
// ===== library: MasterCopy "TimerLibrary" =====

// folder: Timer Library

DATA_BLOCK "TimerLibraryVar"   // DB1
{ S7_Optimized_Access := 'TRUE' }
VERSION : 0.1
   VAR
      POS : Array[0..20] of Struct
         StopMode : Bool;
         ManualMode : Bool;
         AutoMode : Bool;
         CurrentEngineStatus : Int;
         TimeElapsed : Time;
         TimerTime : Time;
         TimerReset : Bool;
         TimerPreset : Bool;
      END_STRUCT;
      HmiPosition : Int := 1;
      ArrayPos : Int;
      Hmi : Struct
         ManualButton : Bool;
         StopButton : Bool;
         AutoButton : Bool;
         TiempoTrans : Time;
      END_STRUCT;
      Temp : Array[0..20] of Struct
         MotorTimer : TP_TIME;
      END_STRUCT;
   END_VAR
BEGIN
   Temp[1].MotorTimer.PT := T#1m;
   Temp[2].MotorTimer.PT := T#2m;
   Temp[3].MotorTimer.PT := T#3m;
   POS[2].TimerTime := T#2m;
   POS[1].TimerTime := T#1m;
   POS[3].TimerTime := T#3m;
END_DATA_BLOCK

FUNCTION "HmiButtonFunction" : Void   // FC4, SCL
{ S7_Optimized_Access := 'TRUE' }
VERSION : 0.1
BEGIN
   (*************************************************************************************************************
                                                 Function Block: Buttons and Operating Modes
   **************************************************************************************************************

   *    Project: Multiple Timer.
   *    Equipment: Siemens S7 1200 PLC
   *    Description: Function and programming of operating modes 
   *    Date: 18/01/2024

   **************************************************************************************************************)


   (* INSERT THIS CODE INTO THE MAIN BLOCK
           "TimerLibraryVar".ArrayPos := "TimerLibraryVar".ArrayPos + 1;
           IF "TimerLibraryVar".ArrayPos > 20 THEN
               "TimerLibraryVar".ArrayPos := 0;
           END_IF;
   *)

   (* INTERFACE NAVIGATION SYSTEM BUTTONS *)

   IF ("TimerLibraryVar".ArrayPos = "TimerLibraryVar".HmiPosition) THEN

       "TimerLibraryVar".POS["TimerLibraryVar".ArrayPos].CurrentEngineStatus := 1;

       IF ("TimerLibraryVar".Hmi.ManualButton) THEN
           "TimerLibraryVar".POS["TimerLibraryVar".ArrayPos].ManualMode := true;
           "TimerLibraryVar".POS["TimerLibraryVar".ArrayPos].StopMode := false;
           "TimerLibraryVar".POS["TimerLibraryVar".ArrayPos].AutoMode := false;
       END_IF;

       IF ("TimerLibraryVar".Hmi.StopButton) THEN
           "TimerLibraryVar".POS["TimerLibraryVar".ArrayPos].ManualMode := false;
           "TimerLibraryVar".POS["TimerLibraryVar".ArrayPos].StopMode := true;
           "TimerLibraryVar".POS["TimerLibraryVar".ArrayPos].AutoMode := false;
       END_IF;

       IF ("TimerLibraryVar".Hmi.AutoButton) THEN
           "TimerLibraryVar".POS["TimerLibraryVar".ArrayPos].ManualMode := false;
           "TimerLibraryVar".POS["TimerLibraryVar".ArrayPos].StopMode := false;
           "TimerLibraryVar".POS["TimerLibraryVar".ArrayPos].AutoMode := true;
       END_IF;
   ELSE
       "TimerLibraryVar".POS["TimerLibraryVar".ArrayPos].CurrentEngineStatus := 0;
   END_IF;

   // END BLOCK
END_FUNCTION

FUNCTION "TimerFunction" : Void   // FC12, SCL
{ S7_Optimized_Access := 'TRUE' }
VERSION : 0.1
BEGIN
   (*************************************************************************************************************
                                                 Function Block: Timer
   **************************************************************************************************************

   *    Project: Multiple Timer.
   *    Equipment: Siemens S7 1200 PLC
   *    Description: Programming the timer function
   *    Date: 18/01/2024

   **************************************************************************************************************)


   "TimerLibraryVar".Temp["TimerLibraryVar".ArrayPos].MotorTimer.TONR(IN := "TimerLibraryVar".POS["TimerLibraryVar".ArrayPos].AutoMode,
                                                                           R := "TimerLibraryVar".POS["TimerLibraryVar".ArrayPos].TimerReset,
                                                                           PT := "TimerLibraryVar".POS["TimerLibraryVar".ArrayPos].TimerTime ,
                                                                           Q=> "TimerLibraryVar".POS["TimerLibraryVar".ArrayPos].TimerPreset,
                                                                           ET => "TimerLibraryVar".POS["TimerLibraryVar".ArrayPos].TimeElapsed);


   // END BLOCK
END_FUNCTION